{attribute 'TcGenerated'}
// This function has been automatically generated from the project information.
VAR_GLOBAL CONSTANT
    {attribute 'const_non_replaced'}
    {attribute 'linkalways'}
    stLibVersion_tmo_lamp_motion : ST_LibVersion := (iMajor := 1, iMinor := 0, iBuild := 4, iRevision := 0, sVersion := '1.0.4');
END_VAR

(* stored: Version 1.1.0.1, ProductVersion 3.1.4022.18
   GVL Global_Version: Id d14ecf09-b76a-4749-bb80-509e26f8448f *)
